FUNCTION_BLOCK RecipeEditor
VAR
	sTitle : STRING;
	sRecipeSteps : ARRAY[1..5] OF STRING;
	pSnapshot : POINTER TO Snapshot;
END_VAR

METHOD createSnapshot : POINTER TO Snapshot
VAR

END_VAR
IF THIS^.pSnapshot <> 0 THEN
	ADSLOGSTR( msgCtrlMask := ADSLOG_MSGTYPE_LOG, msgFmtStr := 'PLC Msg.: %s', strArg := 'Snapshot exists, deleting the old...');
	__DELETE(THIS^.pSnapshot);
END_IF


THIS^.pSnapshot := __NEW(Snapshot(pEditor := ADR(THIS^), sTitle := THIS^.sTitle, sRecipeSteps := THIS^.sRecipeSteps));
createSnapshot := THIS^.pSnapshot;
ADSLOGSTR( msgCtrlMask := ADSLOG_MSGTYPE_LOG, msgFmtStr := 'PLC Msg.: %s', strArg := 'New snapshot generated...');
END_METHOD

METHOD FB_exit : BOOL
VAR_INPUT
	bInCopyCode : BOOL; // if TRUE, the exit method is called for exiting an instance that is copied afterwards (online change).
END_VAR
// Clear the pointer on exit
IF THIS^.pSnapshot <> 0 THEN
	__DELETE(pSnapshot);
END_IF
END_METHOD

METHOD setRecipe
VAR_INPUT
	sRecipeSteps : ARRAY[1..5] OF STRING;
END_VAR
THIS^.sRecipeSteps := sRecipeSteps;
END_METHOD

METHOD setTitle
VAR_INPUT
	sTitle : STRING;
END_VAR
THIS^.sTitle := sTitle;
END_METHOD

END_FUNCTION_BLOCK

(* stored: Version 1.1.0.1, ProductVersion 3.1.4024.12
   POU RecipeEditor: Id {83008406-df84-4944-bf2b-0f186c4ebe1d}, SpecialFunc None
   Method createSnapshot: Id {18292ab5-73b2-4617-81fc-e4aabb59eb99}
   Method FB_exit: Id {8ff35537-a622-442a-a3fe-c602ae73497e}
   Method setRecipe: Id {16ecc6b6-3771-497b-a83c-66283ef3b1d8}
   Method setTitle: Id {39806676-a3dd-40f8-bafc-61a631f38522} *)
